{attribute 'qualified_only'}
//{attribute 'strict'}
{attribute 'to_string'}
TYPE E_MESSAGE_STATE :
(
	MSG_STATE_NULL,
  MSG_STATE_INIT    := 10,
  MSG_STATE_IDLE    := 30,
  MSG_STATE_WRITE   := 50
)UINT;
END_TYPE

(* stored: Version 1.1.0.1
   DUT E_MESSAGE_STATE: Id {df879019-780e-4ea3-8a15-53c86c8a48cd} *)
